FUNCTION_BLOCK Polsador
VAR_INPUT
	Pols:BOOL;
	Reset:BOOL;
END_VAR
VAR_OUTPUT
	Q:BOOL;
END_VAR
VAR
	Estat:BOOL;
	Activa:BOOL;
	Desactiva:BOOL;
	rsEstat:RS;
	Flanc:R_Trig;
	rsEstat2:rs;
END_VAR


Flanc(CLK:=Pols,Q=>Activa);
rsEstat(SET:= (Activa AND NOT Estat), RESET1:= (Activa AND Estat) OR Reset, Q1=>Estat);
Q:=Estat;

END_FUNCTION_BLOCK

(* stored: Version 1.1.0.1, ProductVersion 3.1.4024.11
   POU Polsador: Id {57e842f2-4bf4-4224-bfe8-638a32a2f72d}, SpecialFunc None *)
